// TIA Portal V20 export
DATA_BLOCK "fonction_DB"   // DB2
// stored: MemoryReserve 100, Namespace Ely_2
BEGIN
END_DATA_BLOCK
